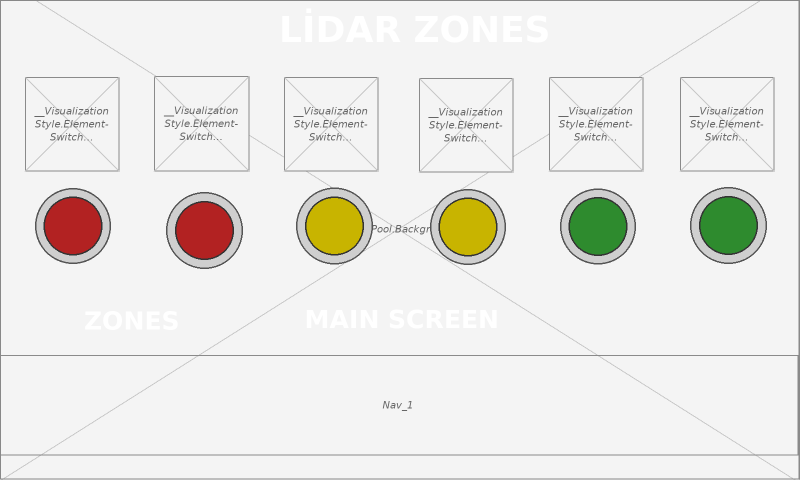
VISUALIZATION Safty_Zones_and_Modes  // 800x480
    Image (-4,-25 804x508), image: ImagePool.Background
    Lamp1 (29,182 88x88), variable: GVLLD.zone_1, invisible if: FALSE, style: Lamp-Lamp1-Red
    Lamp1 (160,182 89x97), variable: GVLLD.zone_2, invisible if: FALSE, style: Lamp-Lamp1-Red
    Lamp1 (290,181 89x90), variable: GVLLD.zone_3, invisible if: FALSE, style: Lamp-Lamp1-Yellow
    Lamp1 (424,182 88x90), variable: GVLLD.zone_4, invisible if: FALSE, style: Lamp-Lamp1-Yellow
    Lamp1 (554,182 88x89), variable: GVLLD.zone_5, invisible if: FALSE, style: Lamp-Lamp1-Green
    Lamp1 (684,181 89x89), tooltip "FALSE", variable: GVLLD.zone_6, style: Lamp-Lamp1-Green
    RoundedRectangle (154,8 522x43), "LİDAR ZONES"
    Frame (-2,355 800x100)
        shows Nav_1()
    Image (680,77 94x94), invisible if: FALSE, input disabled if: FALSE
        OnMouseClick: execute {
            MAIN.Lidar_zones.Front_back_white_zone:= TRUE;
            MAIN.Lidar_zones.Front_back_red_zone:= TRUE;
            MAIN.Lidar_zones.Front_back_purple_zone:= FALSE;
            MAIN.Lidar_zones.Front_back_grey_pink_zone:= FALSE;
            MAIN.zon_1_set:= FALSE;
            MAIN.zon_2_set:= FALSE;
            MAIN.zon_3_set:= FALSE;
            MAIN.zon_4_set:= FALSE;
            MAIN.zon_5_set:= FALSE;
            MAIN.zon_6_set:= TRUE;
        }
    Image (549,77 94x94), invisible if: FALSE, input disabled if: FALSE
        OnMouseClick: execute {
            MAIN.Lidar_zones.Front_back_white_zone:= TRUE;
            MAIN.Lidar_zones.Front_back_red_zone:= FALSE;
            MAIN.Lidar_zones.Front_back_purple_zone:= TRUE;
            MAIN.Lidar_zones.Front_back_grey_pink_zone:= FALSE;
            MAIN.zon_1_set:= FALSE;
            MAIN.zon_2_set:= FALSE;
            MAIN.zon_3_set:= FALSE;
            MAIN.zon_4_set:= FALSE;
            MAIN.zon_5_set:= TRUE;
            MAIN.zon_6_set:= FALSE;
        }
    Image (419,78 94x94), invisible if: FALSE, input disabled if: FALSE
        OnMouseClick: execute {
            MAIN.Lidar_zones.Front_back_white_zone:= FALSE;
            MAIN.Lidar_zones.Front_back_red_zone:= TRUE;
            MAIN.Lidar_zones.Front_back_purple_zone:= TRUE;
            MAIN.Lidar_zones.Front_back_grey_pink_zone:= FALSE;
            MAIN.zon_1_set:= FALSE;
            MAIN.zon_2_set:= FALSE;
            MAIN.zon_3_set:= FALSE;
            MAIN.zon_4_set:= TRUE;
            MAIN.zon_5_set:= FALSE;
            MAIN.zon_6_set:= FALSE;
        }
    Image (284,77 94x94), invisible if: FALSE, input disabled if: FALSE
        OnMouseClick: execute {
            MAIN.Lidar_zones.Front_back_white_zone:= TRUE;
            MAIN.Lidar_zones.Front_back_red_zone:= FALSE;
            MAIN.Lidar_zones.Front_back_purple_zone:= FALSE;
            MAIN.Lidar_zones.Front_back_grey_pink_zone:= TRUE;
            MAIN.zon_1_set:= FALSE;
            MAIN.zon_2_set:= FALSE;
            MAIN.zon_3_set:= TRUE;
            MAIN.zon_4_set:= FALSE;
            MAIN.zon_5_set:= FALSE;
            MAIN.zon_6_set:= FALSE;
        }
    Image (154,76 95x95), invisible if: FALSE, input disabled if: FALSE
        OnMouseClick: execute {
            MAIN.Lidar_zones.Front_back_white_zone:= FALSE;
            MAIN.Lidar_zones.Front_back_red_zone:= TRUE;
            MAIN.Lidar_zones.Front_back_purple_zone:= FALSE;
            MAIN.Lidar_zones.Front_back_grey_pink_zone:= TRUE;
            MAIN.zon_1_set:= FALSE;
            MAIN.zon_2_set:= TRUE;
            MAIN.zon_3_set:= FALSE;
            MAIN.zon_4_set:= FALSE;
            MAIN.zon_5_set:= FALSE;
            MAIN.zon_6_set:= FALSE;
        }
    Image (25,77 94x94), invisible if: FALSE, input disabled if: FALSE
        OnMouseClick: execute {
            MAIN.Lidar_zones.Front_back_white_zone:= FALSE;
            MAIN.Lidar_zones.Front_back_red_zone:= FALSE;
            MAIN.Lidar_zones.Front_back_purple_zone:= TRUE;
            MAIN.Lidar_zones.Front_back_grey_pink_zone:= TRUE;
            MAIN.zon_1_set:= TRUE;
            MAIN.zon_2_set:= FALSE;
            MAIN.zon_3_set:= FALSE;
            MAIN.zon_4_set:= FALSE;
            MAIN.zon_5_set:= FALSE;
            MAIN.zon_6_set:= FALSE;
        }
        OnMouseDown: execute {  }
    RoundedRectangle (286,298 232x42), "MAIN SCREEN"
    RoundedRectangle (15,300 234x41), "ZONES"
END_VISUALIZATION

(* stored: Version 1.1.0.1, ProductVersion 3.1.4024.12
   Visu Safty_Zones_and_Modes: Id {ec5b7dda-c36b-47a6-84d9-79b0592172e2} *)
